TYPE T_OnlineChangeTestCheck :
STRUCT
	bRequired: BOOL;
	bPassed: BOOL;
END_STRUCT
END_TYPE

(* stored: Version 1.1.0.1
   DUT T_OnlineChangeTestCheck: Id {96766ca4-c653-4aa5-b815-a491d940a39e} *)
